// TIA Portal V17 export
// export: Created 2025-03-07T09:18:16.2662316Z, ExportSetting WithDefaults, DisplayName Totally Integrated Automation Portal, DisplayVersion V17 Update 8, DisplayName TIA Portal Openness, DisplayVersion V17 Update 8, DisplayName TIA Portal Version Control Interface, DisplayVersion V17, DisplayName SINAMICS Startdrive Advanced, DisplayVersion V17 SP2, DisplayName SINAMICS Startdrive G110M, G120, G120C, G120D, G120P, G115D, DisplayVersion V17 SP2, DisplayName SINAMICS Startdrive G130, G150, S120, S150, SINAMICS MV, S210, DisplayVersion V17 SP2, DisplayName STEP 7 Professional, DisplayVersion V17 Update 8, DisplayName SINUMERIK ONE STEP 7 Toolbox, DisplayVersion V17 Update 12, DisplayName SINUMERIK 840D sl STEP 7 Toolbox, DisplayVersion V17 Update 12, DisplayName STEP 7 Safety, DisplayVersion V17 Update 6, DisplayName WinCC Advanced, DisplayVersion V17 Update 8
FUNCTION "FC1301_PART_CYCLE_UNIT_03_CLADDING" : Void   // FC1301, LAD
{ S7_Optimized_Access := 'FALSE' }
AUTHOR : ETXETAR
VERSION : 1.0
// stored: AutoNumber false, IsIECCheckEnabled false, SetENOAutomatically false, UDAEnableTagReadback false
   VAR CONSTANT
      FC_NUMBER : DInt := 1301;
   END_VAR
   VAR_TEMP   // added for the SCL form of the ladder/FBD networks
      _w1 : Bool;
      _w2 : Bool;
   END_VAR
BEGIN

REGION Network 1: GENERAL CONDITIONS
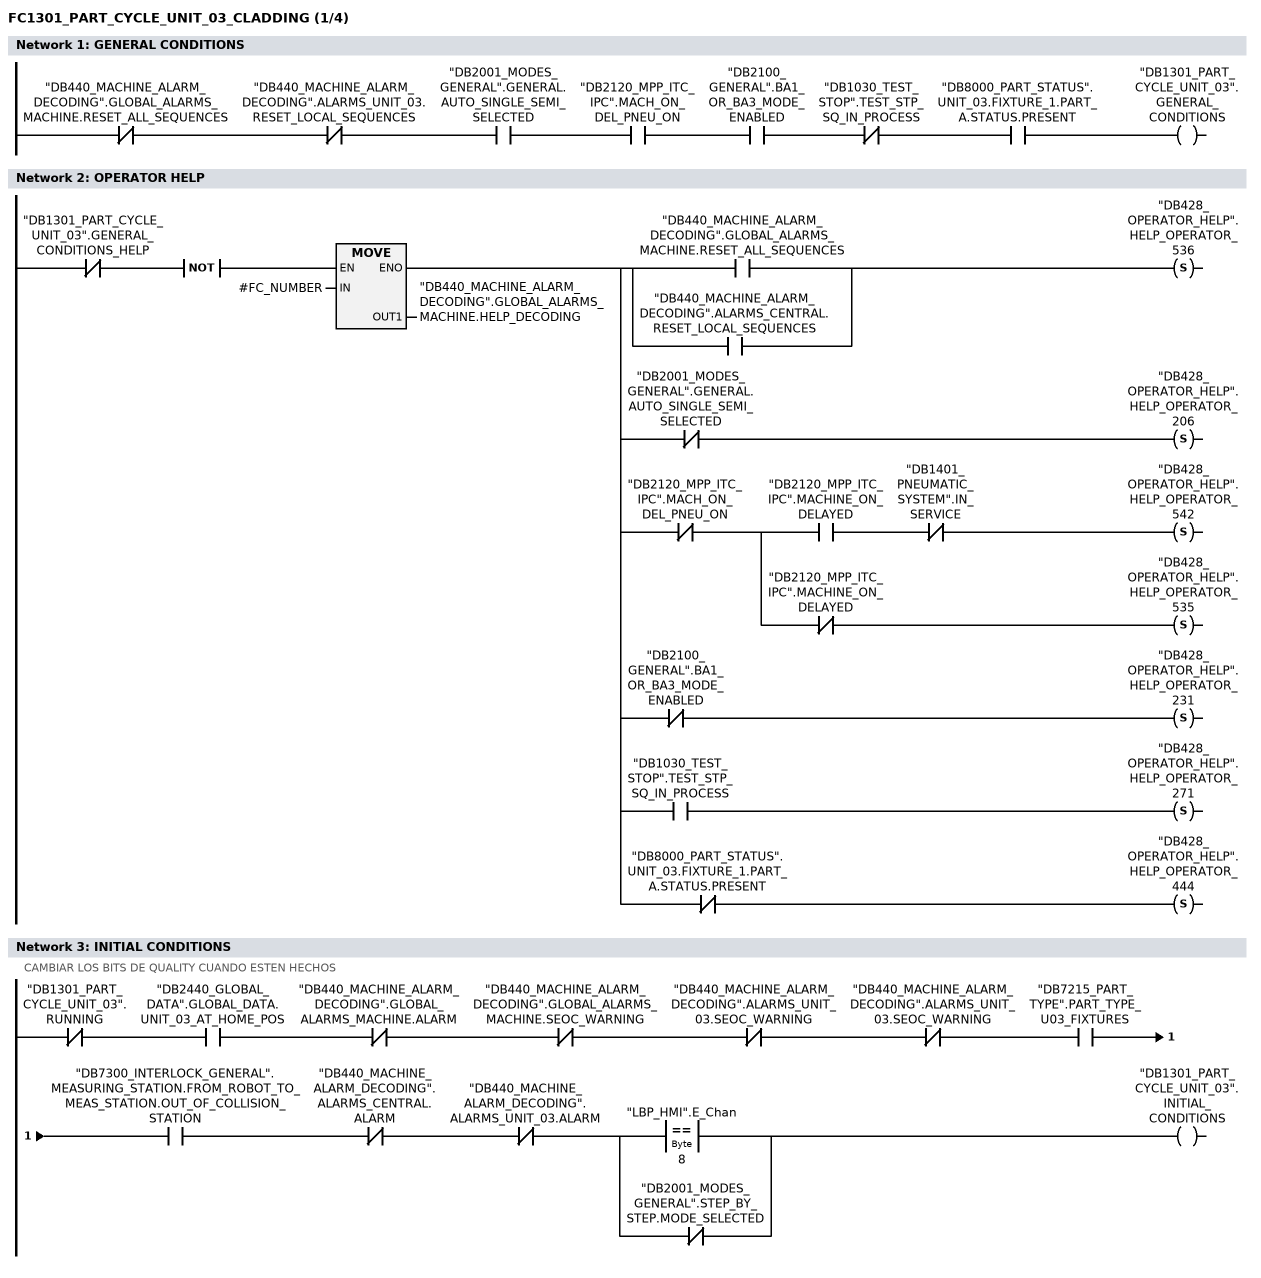
   RUNG wire#powerrail
      I_Contact( "DB440_MACHINE_ALARM_DECODING".GLOBAL_ALARMS_MACHINE.RESET_ALL_SEQUENCES )
      I_Contact( "DB440_MACHINE_ALARM_DECODING".ALARMS_UNIT_03.RESET_LOCAL_SEQUENCES )
      Contact( "DB2001_MODES_GENERAL".GENERAL.AUTO_SINGLE_SEMI_SELECTED )
      Contact( "DB2120_MPP_ITC_IPC".MACH_ON_DEL_PNEU_ON )
      Contact( "DB2100_GENERAL".BA1_OR_BA3_MODE_ENABLED )
      I_Contact( "DB1030_TEST_STOP".TEST_STP_SQ_IN_PROCESS )
      Contact( "DB8000_PART_STATUS".UNIT_03.FIXTURE_1.PART_A.STATUS.PRESENT )
      Coil( "DB1301_PART_CYCLE_UNIT_03".GENERAL_CONDITIONS )
   END_RUNG
   // the same network as SCL:
   "DB1301_PART_CYCLE_UNIT_03".GENERAL_CONDITIONS := NOT "DB440_MACHINE_ALARM_DECODING".GLOBAL_ALARMS_MACHINE.RESET_ALL_SEQUENCES AND NOT "DB440_MACHINE_ALARM_DECODING".ALARMS_UNIT_03.RESET_LOCAL_SEQUENCES AND "DB2001_MODES_GENERAL".GENERAL.AUTO_SINGLE_SEMI_SELECTED AND "DB2120_MPP_ITC_IPC".MACH_ON_DEL_PNEU_ON AND "DB2100_GENERAL".BA1_OR_BA3_MODE_ENABLED AND NOT "DB1030_TEST_STOP".TEST_STP_SQ_IN_PROCESS AND "DB8000_PART_STATUS".UNIT_03.FIXTURE_1.PART_A.STATUS.PRESENT;
END_REGION

REGION Network 2: OPERATOR HELP
   RUNG wire#powerrail
      I_Contact( "DB1301_PART_CYCLE_UNIT_03".GENERAL_CONDITIONS_HELP )
      Not()
      { S7_GenerateENO := "TRUE" } Move(in := #FC_NUMBER, out1 => "DB440_MACHINE_ALARM_DECODING".GLOBAL_ALARMS_MACHINE.HELP_DECODING)
      wire#w1
      Contact( "DB440_MACHINE_ALARM_DECODING".GLOBAL_ALARMS_MACHINE.RESET_ALL_SEQUENCES )
      wire#w2
      S_Coil( "DB428_OPERATOR_HELP".HELP_OPERATOR_536 )
   END_RUNG
   RUNG wire#w1
      Contact( "DB440_MACHINE_ALARM_DECODING".ALARMS_CENTRAL.RESET_LOCAL_SEQUENCES )
   END_RUNG wire#w2
   RUNG wire#w1
      I_Contact( "DB2001_MODES_GENERAL".GENERAL.AUTO_SINGLE_SEMI_SELECTED )
      S_Coil( "DB428_OPERATOR_HELP".HELP_OPERATOR_206 )
   END_RUNG
   RUNG wire#w1
      I_Contact( "DB2120_MPP_ITC_IPC".MACH_ON_DEL_PNEU_ON )
      wire#w3
      Contact( "DB2120_MPP_ITC_IPC".MACHINE_ON_DELAYED )
      I_Contact( "DB1401_PNEUMATIC_SYSTEM".IN_SERVICE )
      S_Coil( "DB428_OPERATOR_HELP".HELP_OPERATOR_542 )
   END_RUNG
   RUNG wire#w3
      I_Contact( "DB2120_MPP_ITC_IPC".MACHINE_ON_DELAYED )
      S_Coil( "DB428_OPERATOR_HELP".HELP_OPERATOR_535 )
   END_RUNG
   RUNG wire#w1
      I_Contact( "DB2100_GENERAL".BA1_OR_BA3_MODE_ENABLED )
      S_Coil( "DB428_OPERATOR_HELP".HELP_OPERATOR_231 )
   END_RUNG
   RUNG wire#w1
      Contact( "DB1030_TEST_STOP".TEST_STP_SQ_IN_PROCESS )
      S_Coil( "DB428_OPERATOR_HELP".HELP_OPERATOR_271 )
   END_RUNG
   RUNG wire#w1
      I_Contact( "DB8000_PART_STATUS".UNIT_03.FIXTURE_1.PART_A.STATUS.PRESENT )
      S_Coil( "DB428_OPERATOR_HELP".HELP_OPERATOR_444 )
   END_RUNG
   // the same network as SCL:
   // ENO of a box is taken as its EN; it also drops when the box reports an error
   #_w1 := NOT (NOT "DB1301_PART_CYCLE_UNIT_03".GENERAL_CONDITIONS_HELP);
   IF #_w1 THEN "DB440_MACHINE_ALARM_DECODING".GLOBAL_ALARMS_MACHINE.HELP_DECODING := #FC_NUMBER; END_IF;
   IF #_w1 AND ("DB440_MACHINE_ALARM_DECODING".GLOBAL_ALARMS_MACHINE.RESET_ALL_SEQUENCES OR "DB440_MACHINE_ALARM_DECODING".ALARMS_CENTRAL.RESET_LOCAL_SEQUENCES) THEN
       "DB428_OPERATOR_HELP".HELP_OPERATOR_536 := TRUE;
   END_IF;
   IF #_w1 AND NOT "DB2001_MODES_GENERAL".GENERAL.AUTO_SINGLE_SEMI_SELECTED THEN
       "DB428_OPERATOR_HELP".HELP_OPERATOR_206 := TRUE;
   END_IF;
   #_w2 := #_w1 AND NOT "DB2120_MPP_ITC_IPC".MACH_ON_DEL_PNEU_ON;
   IF #_w2 AND "DB2120_MPP_ITC_IPC".MACHINE_ON_DELAYED AND NOT "DB1401_PNEUMATIC_SYSTEM".IN_SERVICE THEN
       "DB428_OPERATOR_HELP".HELP_OPERATOR_542 := TRUE;
   END_IF;
   IF #_w2 AND NOT "DB2120_MPP_ITC_IPC".MACHINE_ON_DELAYED THEN
       "DB428_OPERATOR_HELP".HELP_OPERATOR_535 := TRUE;
   END_IF;
   IF #_w1 AND NOT "DB2100_GENERAL".BA1_OR_BA3_MODE_ENABLED THEN
       "DB428_OPERATOR_HELP".HELP_OPERATOR_231 := TRUE;
   END_IF;
   IF #_w1 AND "DB1030_TEST_STOP".TEST_STP_SQ_IN_PROCESS THEN
       "DB428_OPERATOR_HELP".HELP_OPERATOR_271 := TRUE;
   END_IF;
   IF #_w1 AND NOT "DB8000_PART_STATUS".UNIT_03.FIXTURE_1.PART_A.STATUS.PRESENT THEN
       "DB428_OPERATOR_HELP".HELP_OPERATOR_444 := TRUE;
   END_IF;
END_REGION

REGION Network 3: INITIAL CONDITIONS
   // CAMBIAR LOS BITS DE QUALITY CUANDO ESTEN HECHOS
   RUNG wire#powerrail
      I_Contact( "DB1301_PART_CYCLE_UNIT_03".RUNNING )
      Contact( "DB2440_GLOBAL_DATA".GLOBAL_DATA.UNIT_03_AT_HOME_POS )
      I_Contact( "DB440_MACHINE_ALARM_DECODING".GLOBAL_ALARMS_MACHINE.ALARM )
      I_Contact( "DB440_MACHINE_ALARM_DECODING".GLOBAL_ALARMS_MACHINE.SEOC_WARNING )
      I_Contact( "DB440_MACHINE_ALARM_DECODING".ALARMS_UNIT_03.SEOC_WARNING )
      I_Contact( "DB440_MACHINE_ALARM_DECODING".ALARMS_UNIT_03.SEOC_WARNING )
      Contact( "DB7215_PART_TYPE".PART_TYPE_U03_FIXTURES )
      Contact( "DB7300_INTERLOCK_GENERAL".MEASURING_STATION.FROM_ROBOT_TO_MEAS_STATION.OUT_OF_COLLISION_STATION )
      I_Contact( "DB440_MACHINE_ALARM_DECODING".ALARMS_CENTRAL.ALARM )
      I_Contact( "DB440_MACHINE_ALARM_DECODING".ALARMS_UNIT_03.ALARM )
      wire#w1
      { S7_Templates := "SrcType := Byte" } EQ_Contact(in1 := "LBP_HMI".E_Chan, in2 := 8)
      wire#w2
      Coil( "DB1301_PART_CYCLE_UNIT_03".INITIAL_CONDITIONS )
   END_RUNG
   RUNG wire#w1
      I_Contact( "DB2001_MODES_GENERAL".STEP_BY_STEP.MODE_SELECTED )
   END_RUNG wire#w2
   // the same network as SCL:
   "DB1301_PART_CYCLE_UNIT_03".INITIAL_CONDITIONS := NOT "DB1301_PART_CYCLE_UNIT_03".RUNNING AND "DB2440_GLOBAL_DATA".GLOBAL_DATA.UNIT_03_AT_HOME_POS AND NOT "DB440_MACHINE_ALARM_DECODING".GLOBAL_ALARMS_MACHINE.ALARM AND NOT "DB440_MACHINE_ALARM_DECODING".GLOBAL_ALARMS_MACHINE.SEOC_WARNING AND NOT "DB440_MACHINE_ALARM_DECODING".ALARMS_UNIT_03.SEOC_WARNING AND NOT "DB440_MACHINE_ALARM_DECODING".ALARMS_UNIT_03.SEOC_WARNING AND "DB7215_PART_TYPE".PART_TYPE_U03_FIXTURES AND "DB7300_INTERLOCK_GENERAL".MEASURING_STATION.FROM_ROBOT_TO_MEAS_STATION.OUT_OF_COLLISION_STATION AND NOT "DB440_MACHINE_ALARM_DECODING".ALARMS_CENTRAL.ALARM AND NOT "DB440_MACHINE_ALARM_DECODING".ALARMS_UNIT_03.ALARM AND (("LBP_HMI".E_Chan = 8) OR NOT "DB2001_MODES_GENERAL".STEP_BY_STEP.MODE_SELECTED);
END_REGION

REGION Network 4: OPERATOR HELP
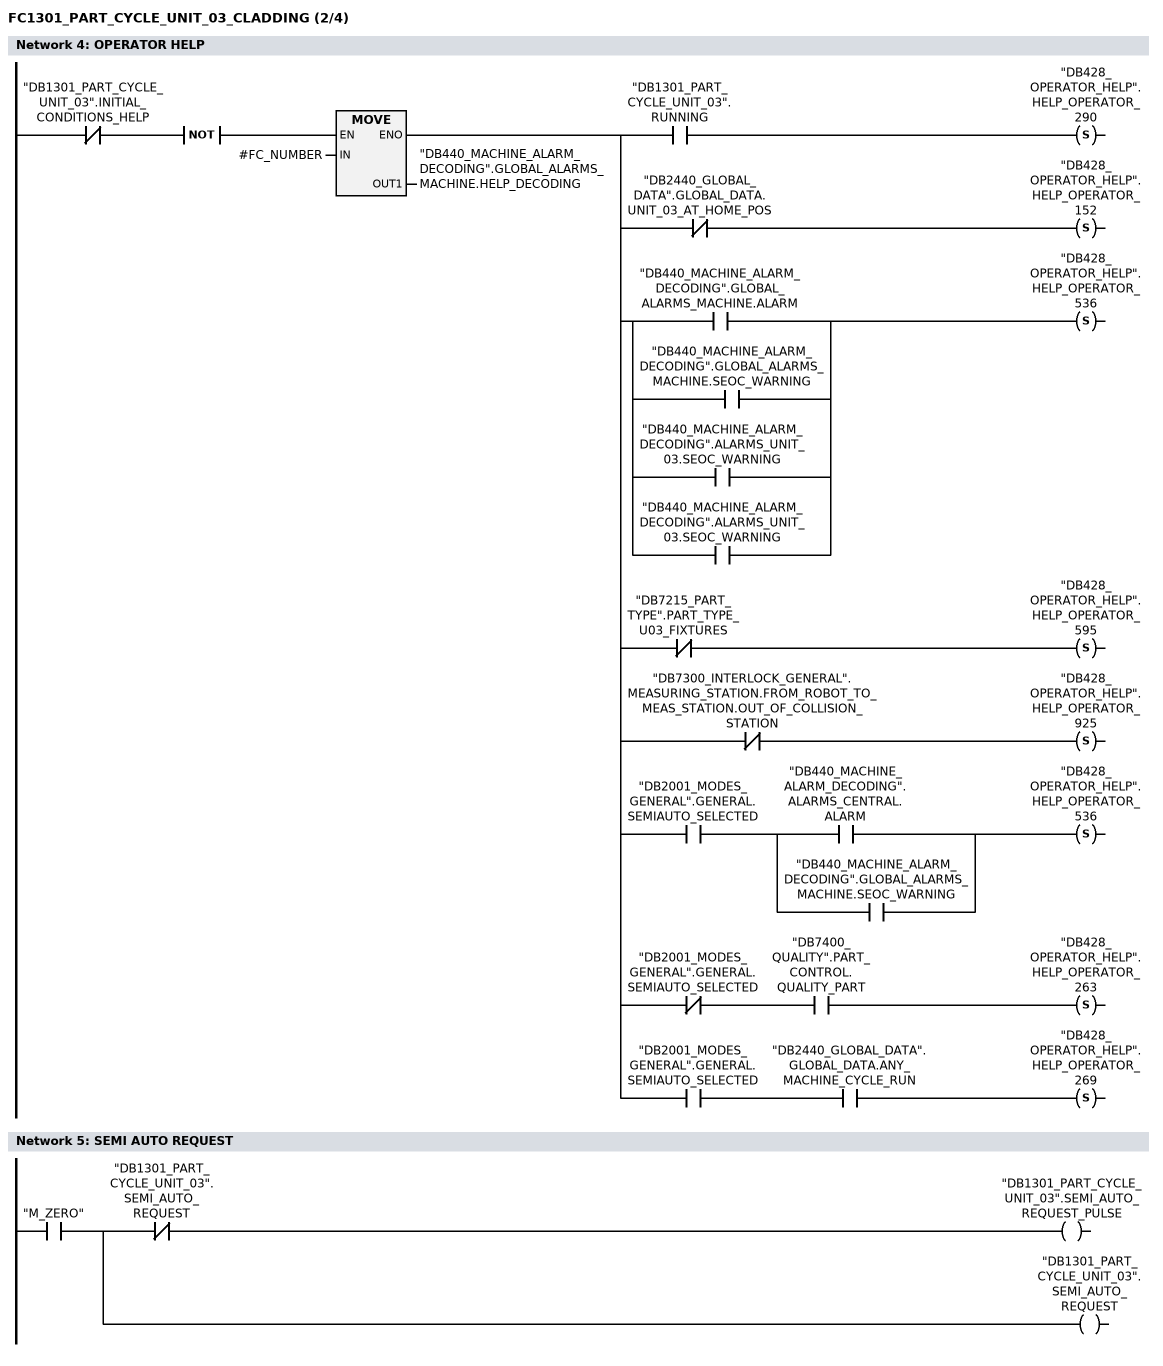
   RUNG wire#powerrail
      I_Contact( "DB1301_PART_CYCLE_UNIT_03".INITIAL_CONDITIONS_HELP )
      Not()
      { S7_GenerateENO := "TRUE" } Move(in := #FC_NUMBER, out1 => "DB440_MACHINE_ALARM_DECODING".GLOBAL_ALARMS_MACHINE.HELP_DECODING)
      wire#w1
      Contact( "DB1301_PART_CYCLE_UNIT_03".RUNNING )
      S_Coil( "DB428_OPERATOR_HELP".HELP_OPERATOR_290 )
   END_RUNG
   RUNG wire#w1
      I_Contact( "DB2440_GLOBAL_DATA".GLOBAL_DATA.UNIT_03_AT_HOME_POS )
      S_Coil( "DB428_OPERATOR_HELP".HELP_OPERATOR_152 )
   END_RUNG
   RUNG wire#w1
      Contact( "DB440_MACHINE_ALARM_DECODING".GLOBAL_ALARMS_MACHINE.ALARM )
      wire#w2
      S_Coil( "DB428_OPERATOR_HELP".HELP_OPERATOR_536 )
   END_RUNG
   RUNG wire#w1
      Contact( "DB440_MACHINE_ALARM_DECODING".GLOBAL_ALARMS_MACHINE.SEOC_WARNING )
   END_RUNG wire#w2
   RUNG wire#w1
      Contact( "DB440_MACHINE_ALARM_DECODING".ALARMS_UNIT_03.SEOC_WARNING )
   END_RUNG wire#w2
   RUNG wire#w1
      Contact( "DB440_MACHINE_ALARM_DECODING".ALARMS_UNIT_03.SEOC_WARNING )
   END_RUNG wire#w2
   RUNG wire#w1
      I_Contact( "DB7215_PART_TYPE".PART_TYPE_U03_FIXTURES )
      S_Coil( "DB428_OPERATOR_HELP".HELP_OPERATOR_595 )
   END_RUNG
   RUNG wire#w1
      I_Contact( "DB7300_INTERLOCK_GENERAL".MEASURING_STATION.FROM_ROBOT_TO_MEAS_STATION.OUT_OF_COLLISION_STATION )
      S_Coil( "DB428_OPERATOR_HELP".HELP_OPERATOR_925 )
   END_RUNG
   RUNG wire#w1
      Contact( "DB2001_MODES_GENERAL".GENERAL.SEMIAUTO_SELECTED )
      wire#w3
      Contact( "DB440_MACHINE_ALARM_DECODING".ALARMS_CENTRAL.ALARM )
      wire#w4
      S_Coil( "DB428_OPERATOR_HELP".HELP_OPERATOR_536 )
   END_RUNG
   RUNG wire#w3
      Contact( "DB440_MACHINE_ALARM_DECODING".GLOBAL_ALARMS_MACHINE.SEOC_WARNING )
   END_RUNG wire#w4
   RUNG wire#w1
      I_Contact( "DB2001_MODES_GENERAL".GENERAL.SEMIAUTO_SELECTED )
      Contact( "DB7400_QUALITY".PART_CONTROL.QUALITY_PART )
      S_Coil( "DB428_OPERATOR_HELP".HELP_OPERATOR_263 )
   END_RUNG
   RUNG wire#w1
      Contact( "DB2001_MODES_GENERAL".GENERAL.SEMIAUTO_SELECTED )
      Contact( "DB2440_GLOBAL_DATA".GLOBAL_DATA.ANY_MACHINE_CYCLE_RUN )
      S_Coil( "DB428_OPERATOR_HELP".HELP_OPERATOR_269 )
   END_RUNG
   // the same network as SCL:
   // ENO of a box is taken as its EN; it also drops when the box reports an error
   #_w1 := NOT (NOT "DB1301_PART_CYCLE_UNIT_03".INITIAL_CONDITIONS_HELP);
   IF #_w1 THEN "DB440_MACHINE_ALARM_DECODING".GLOBAL_ALARMS_MACHINE.HELP_DECODING := #FC_NUMBER; END_IF;
   IF #_w1 AND "DB1301_PART_CYCLE_UNIT_03".RUNNING THEN
       "DB428_OPERATOR_HELP".HELP_OPERATOR_290 := TRUE;
   END_IF;
   IF #_w1 AND NOT "DB2440_GLOBAL_DATA".GLOBAL_DATA.UNIT_03_AT_HOME_POS THEN
       "DB428_OPERATOR_HELP".HELP_OPERATOR_152 := TRUE;
   END_IF;
   IF #_w1 AND ("DB440_MACHINE_ALARM_DECODING".GLOBAL_ALARMS_MACHINE.ALARM OR "DB440_MACHINE_ALARM_DECODING".GLOBAL_ALARMS_MACHINE.SEOC_WARNING OR "DB440_MACHINE_ALARM_DECODING".ALARMS_UNIT_03.SEOC_WARNING OR "DB440_MACHINE_ALARM_DECODING".ALARMS_UNIT_03.SEOC_WARNING) THEN
       "DB428_OPERATOR_HELP".HELP_OPERATOR_536 := TRUE;
   END_IF;
   IF #_w1 AND NOT "DB7215_PART_TYPE".PART_TYPE_U03_FIXTURES THEN
       "DB428_OPERATOR_HELP".HELP_OPERATOR_595 := TRUE;
   END_IF;
   IF #_w1 AND NOT "DB7300_INTERLOCK_GENERAL".MEASURING_STATION.FROM_ROBOT_TO_MEAS_STATION.OUT_OF_COLLISION_STATION THEN
       "DB428_OPERATOR_HELP".HELP_OPERATOR_925 := TRUE;
   END_IF;
   IF #_w1 AND "DB2001_MODES_GENERAL".GENERAL.SEMIAUTO_SELECTED AND ("DB440_MACHINE_ALARM_DECODING".ALARMS_CENTRAL.ALARM OR "DB440_MACHINE_ALARM_DECODING".GLOBAL_ALARMS_MACHINE.SEOC_WARNING) THEN
       "DB428_OPERATOR_HELP".HELP_OPERATOR_536 := TRUE;
   END_IF;
   IF #_w1 AND NOT "DB2001_MODES_GENERAL".GENERAL.SEMIAUTO_SELECTED AND "DB7400_QUALITY".PART_CONTROL.QUALITY_PART THEN
       "DB428_OPERATOR_HELP".HELP_OPERATOR_263 := TRUE;
   END_IF;
   IF #_w1 AND "DB2001_MODES_GENERAL".GENERAL.SEMIAUTO_SELECTED AND "DB2440_GLOBAL_DATA".GLOBAL_DATA.ANY_MACHINE_CYCLE_RUN THEN
       "DB428_OPERATOR_HELP".HELP_OPERATOR_269 := TRUE;
   END_IF;
END_REGION

REGION Network 5: SEMI AUTO REQUEST
   RUNG wire#powerrail
      Contact( "M_ZERO" )
      wire#w1
      I_Contact( "DB1301_PART_CYCLE_UNIT_03".SEMI_AUTO_REQUEST )
      Coil( "DB1301_PART_CYCLE_UNIT_03".SEMI_AUTO_REQUEST_PULSE )
   END_RUNG
   RUNG wire#w1
      Coil( "DB1301_PART_CYCLE_UNIT_03".SEMI_AUTO_REQUEST )
   END_RUNG
   // the same network as SCL:
   "DB1301_PART_CYCLE_UNIT_03".SEMI_AUTO_REQUEST_PULSE := "M_ZERO" AND NOT "DB1301_PART_CYCLE_UNIT_03".SEMI_AUTO_REQUEST;
   "DB1301_PART_CYCLE_UNIT_03".SEMI_AUTO_REQUEST := "M_ZERO";
END_REGION

REGION Network 6: OPERATOR HELP
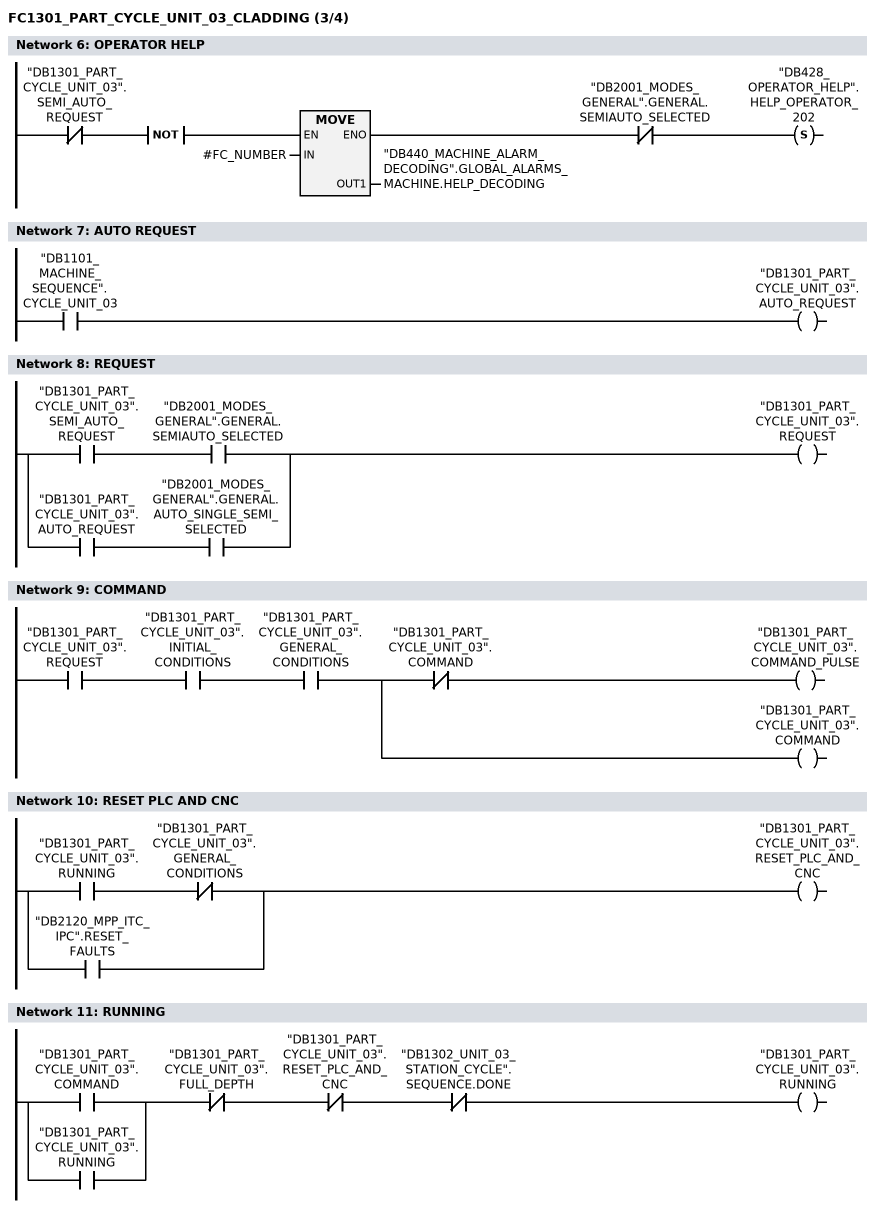
   RUNG wire#powerrail
      I_Contact( "DB1301_PART_CYCLE_UNIT_03".SEMI_AUTO_REQUEST )
      Not()
      { S7_GenerateENO := "TRUE" } Move(in := #FC_NUMBER, out1 => "DB440_MACHINE_ALARM_DECODING".GLOBAL_ALARMS_MACHINE.HELP_DECODING)
      I_Contact( "DB2001_MODES_GENERAL".GENERAL.SEMIAUTO_SELECTED )
      S_Coil( "DB428_OPERATOR_HELP".HELP_OPERATOR_202 )
   END_RUNG
   // the same network as SCL:
   // ENO of a box is taken as its EN; it also drops when the box reports an error
   #_w1 := NOT (NOT "DB1301_PART_CYCLE_UNIT_03".SEMI_AUTO_REQUEST);
   IF #_w1 THEN "DB440_MACHINE_ALARM_DECODING".GLOBAL_ALARMS_MACHINE.HELP_DECODING := #FC_NUMBER; END_IF;
   IF #_w1 AND NOT "DB2001_MODES_GENERAL".GENERAL.SEMIAUTO_SELECTED THEN
       "DB428_OPERATOR_HELP".HELP_OPERATOR_202 := TRUE;
   END_IF;
END_REGION

REGION Network 7: AUTO REQUEST
   RUNG wire#powerrail
      Contact( "DB1101_MACHINE_SEQUENCE".CYCLE_UNIT_03 )
      Coil( "DB1301_PART_CYCLE_UNIT_03".AUTO_REQUEST )
   END_RUNG
   // the same network as SCL:
   "DB1301_PART_CYCLE_UNIT_03".AUTO_REQUEST := "DB1101_MACHINE_SEQUENCE".CYCLE_UNIT_03;
END_REGION

REGION Network 8: REQUEST
   RUNG wire#powerrail
      Contact( "DB1301_PART_CYCLE_UNIT_03".SEMI_AUTO_REQUEST )
      Contact( "DB2001_MODES_GENERAL".GENERAL.SEMIAUTO_SELECTED )
      wire#w1
      Coil( "DB1301_PART_CYCLE_UNIT_03".REQUEST )
   END_RUNG
   RUNG wire#powerrail
      Contact( "DB1301_PART_CYCLE_UNIT_03".AUTO_REQUEST )
      Contact( "DB2001_MODES_GENERAL".GENERAL.AUTO_SINGLE_SEMI_SELECTED )
   END_RUNG wire#w1
   // the same network as SCL:
   "DB1301_PART_CYCLE_UNIT_03".REQUEST := ("DB1301_PART_CYCLE_UNIT_03".SEMI_AUTO_REQUEST AND "DB2001_MODES_GENERAL".GENERAL.SEMIAUTO_SELECTED) OR ("DB1301_PART_CYCLE_UNIT_03".AUTO_REQUEST AND "DB2001_MODES_GENERAL".GENERAL.AUTO_SINGLE_SEMI_SELECTED);
END_REGION

REGION Network 9: COMMAND
   RUNG wire#powerrail
      Contact( "DB1301_PART_CYCLE_UNIT_03".REQUEST )
      Contact( "DB1301_PART_CYCLE_UNIT_03".INITIAL_CONDITIONS )
      Contact( "DB1301_PART_CYCLE_UNIT_03".GENERAL_CONDITIONS )
      wire#w1
      I_Contact( "DB1301_PART_CYCLE_UNIT_03".COMMAND )
      Coil( "DB1301_PART_CYCLE_UNIT_03".COMMAND_PULSE )
   END_RUNG
   RUNG wire#w1
      Coil( "DB1301_PART_CYCLE_UNIT_03".COMMAND )
   END_RUNG
   // the same network as SCL:
   #_w1 := "DB1301_PART_CYCLE_UNIT_03".REQUEST AND "DB1301_PART_CYCLE_UNIT_03".INITIAL_CONDITIONS AND "DB1301_PART_CYCLE_UNIT_03".GENERAL_CONDITIONS;
   "DB1301_PART_CYCLE_UNIT_03".COMMAND_PULSE := #_w1 AND NOT "DB1301_PART_CYCLE_UNIT_03".COMMAND;
   "DB1301_PART_CYCLE_UNIT_03".COMMAND := #_w1;
END_REGION

REGION Network 10: RESET PLC AND CNC
   RUNG wire#powerrail
      Contact( "DB1301_PART_CYCLE_UNIT_03".RUNNING )
      I_Contact( "DB1301_PART_CYCLE_UNIT_03".GENERAL_CONDITIONS )
      wire#w1
      Coil( "DB1301_PART_CYCLE_UNIT_03".RESET_PLC_AND_CNC )
   END_RUNG
   RUNG wire#powerrail
      Contact( "DB2120_MPP_ITC_IPC".RESET_FAULTS )
   END_RUNG wire#w1
   // the same network as SCL:
   "DB1301_PART_CYCLE_UNIT_03".RESET_PLC_AND_CNC := ("DB1301_PART_CYCLE_UNIT_03".RUNNING AND NOT "DB1301_PART_CYCLE_UNIT_03".GENERAL_CONDITIONS) OR "DB2120_MPP_ITC_IPC".RESET_FAULTS;
END_REGION

REGION Network 11: RUNNING
   RUNG wire#powerrail
      Contact( "DB1301_PART_CYCLE_UNIT_03".COMMAND )
      wire#w1
      I_Contact( "DB1301_PART_CYCLE_UNIT_03".FULL_DEPTH )
      I_Contact( "DB1301_PART_CYCLE_UNIT_03".RESET_PLC_AND_CNC )
      I_Contact( "DB1302_UNIT_03_STATION_CYCLE".SEQUENCE.DONE )
      Coil( "DB1301_PART_CYCLE_UNIT_03".RUNNING )
   END_RUNG
   RUNG wire#powerrail
      Contact( "DB1301_PART_CYCLE_UNIT_03".RUNNING )
   END_RUNG wire#w1
   // the same network as SCL:
   "DB1301_PART_CYCLE_UNIT_03".RUNNING := ("DB1301_PART_CYCLE_UNIT_03".COMMAND OR "DB1301_PART_CYCLE_UNIT_03".RUNNING) AND NOT "DB1301_PART_CYCLE_UNIT_03".FULL_DEPTH AND NOT "DB1301_PART_CYCLE_UNIT_03".RESET_PLC_AND_CNC AND NOT "DB1302_UNIT_03_STATION_CYCLE".SEQUENCE.DONE;
END_REGION

REGION Network 12: CYCLE MEASURE UNIT STATION
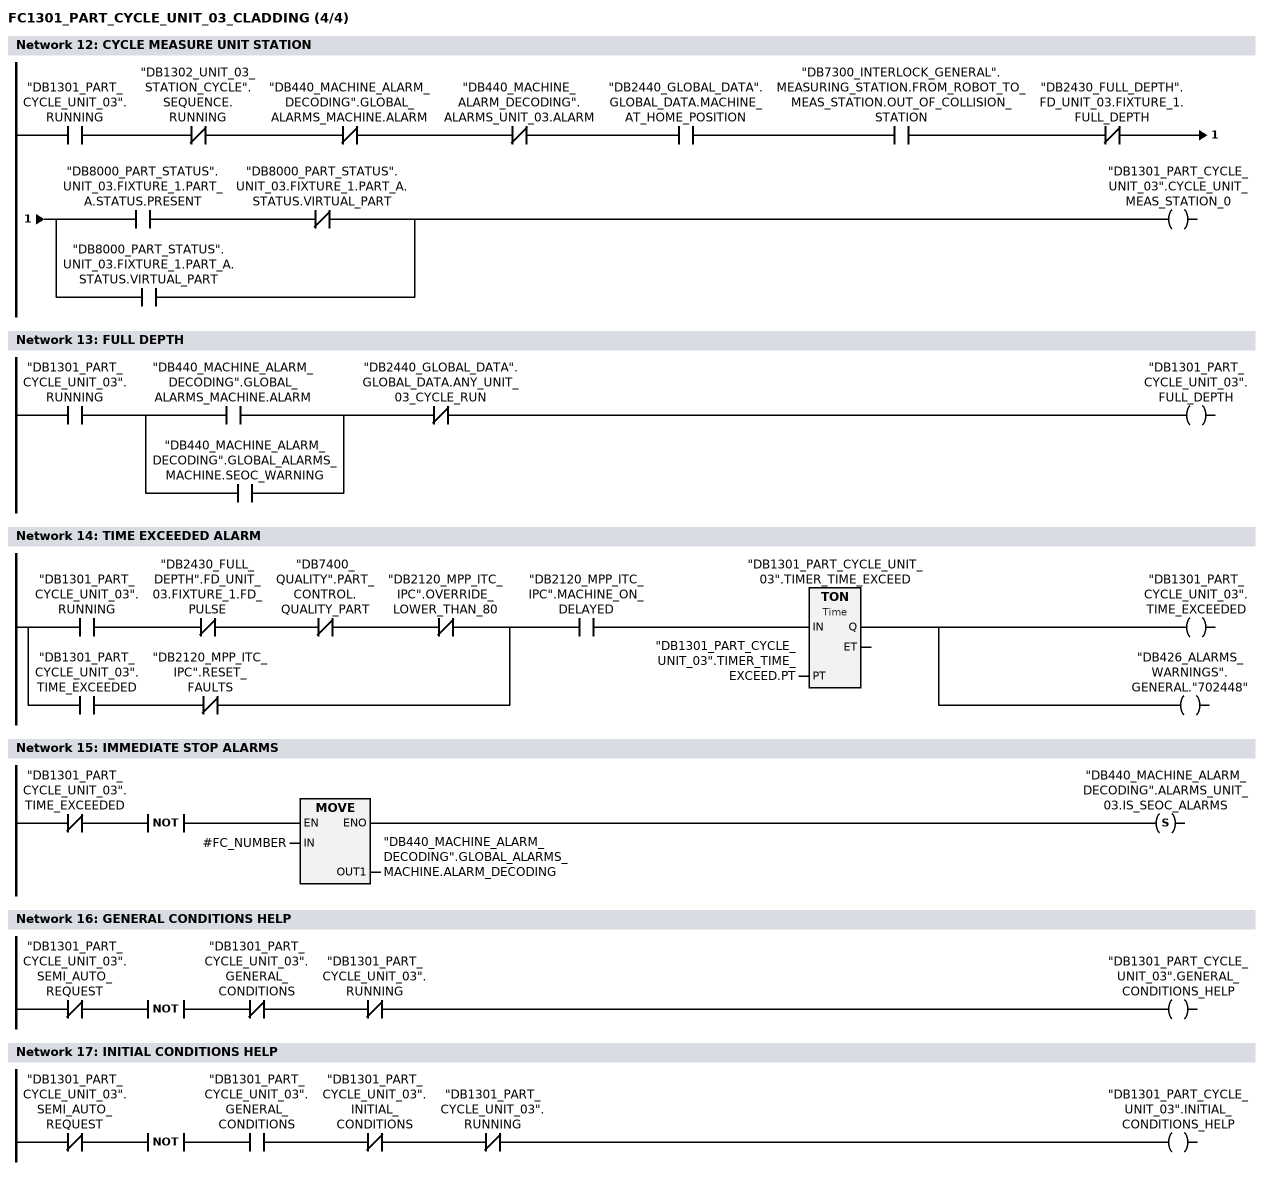
   RUNG wire#powerrail
      Contact( "DB1301_PART_CYCLE_UNIT_03".RUNNING )
      I_Contact( "DB1302_UNIT_03_STATION_CYCLE".SEQUENCE.RUNNING )
      I_Contact( "DB440_MACHINE_ALARM_DECODING".GLOBAL_ALARMS_MACHINE.ALARM )
      I_Contact( "DB440_MACHINE_ALARM_DECODING".ALARMS_UNIT_03.ALARM )
      Contact( "DB2440_GLOBAL_DATA".GLOBAL_DATA.MACHINE_AT_HOME_POSITION )
      Contact( "DB7300_INTERLOCK_GENERAL".MEASURING_STATION.FROM_ROBOT_TO_MEAS_STATION.OUT_OF_COLLISION_STATION )
      I_Contact( "DB2430_FULL_DEPTH".FD_UNIT_03.FIXTURE_1.FULL_DEPTH )
      wire#w1
      Contact( "DB8000_PART_STATUS".UNIT_03.FIXTURE_1.PART_A.STATUS.PRESENT )
      I_Contact( "DB8000_PART_STATUS".UNIT_03.FIXTURE_1.PART_A.STATUS.VIRTUAL_PART )
      wire#w2
      Coil( "DB1301_PART_CYCLE_UNIT_03".CYCLE_UNIT_MEAS_STATION_0 )
   END_RUNG
   RUNG wire#w1
      Contact( "DB8000_PART_STATUS".UNIT_03.FIXTURE_1.PART_A.STATUS.VIRTUAL_PART )
   END_RUNG wire#w2
   // the same network as SCL:
   "DB1301_PART_CYCLE_UNIT_03".CYCLE_UNIT_MEAS_STATION_0 := "DB1301_PART_CYCLE_UNIT_03".RUNNING AND NOT "DB1302_UNIT_03_STATION_CYCLE".SEQUENCE.RUNNING AND NOT "DB440_MACHINE_ALARM_DECODING".GLOBAL_ALARMS_MACHINE.ALARM AND NOT "DB440_MACHINE_ALARM_DECODING".ALARMS_UNIT_03.ALARM AND "DB2440_GLOBAL_DATA".GLOBAL_DATA.MACHINE_AT_HOME_POSITION AND "DB7300_INTERLOCK_GENERAL".MEASURING_STATION.FROM_ROBOT_TO_MEAS_STATION.OUT_OF_COLLISION_STATION AND NOT "DB2430_FULL_DEPTH".FD_UNIT_03.FIXTURE_1.FULL_DEPTH AND (("DB8000_PART_STATUS".UNIT_03.FIXTURE_1.PART_A.STATUS.PRESENT AND NOT "DB8000_PART_STATUS".UNIT_03.FIXTURE_1.PART_A.STATUS.VIRTUAL_PART) OR "DB8000_PART_STATUS".UNIT_03.FIXTURE_1.PART_A.STATUS.VIRTUAL_PART);
END_REGION

REGION Network 13: FULL DEPTH
   RUNG wire#powerrail
      Contact( "DB1301_PART_CYCLE_UNIT_03".RUNNING )
      wire#w1
      Contact( "DB440_MACHINE_ALARM_DECODING".GLOBAL_ALARMS_MACHINE.ALARM )
      wire#w2
      I_Contact( "DB2440_GLOBAL_DATA".GLOBAL_DATA.ANY_UNIT_03_CYCLE_RUN )
      Coil( "DB1301_PART_CYCLE_UNIT_03".FULL_DEPTH )
   END_RUNG
   RUNG wire#w1
      Contact( "DB440_MACHINE_ALARM_DECODING".GLOBAL_ALARMS_MACHINE.SEOC_WARNING )
   END_RUNG wire#w2
   // the same network as SCL:
   "DB1301_PART_CYCLE_UNIT_03".FULL_DEPTH := "DB1301_PART_CYCLE_UNIT_03".RUNNING AND ("DB440_MACHINE_ALARM_DECODING".GLOBAL_ALARMS_MACHINE.ALARM OR "DB440_MACHINE_ALARM_DECODING".GLOBAL_ALARMS_MACHINE.SEOC_WARNING) AND NOT "DB2440_GLOBAL_DATA".GLOBAL_DATA.ANY_UNIT_03_CYCLE_RUN;
END_REGION

REGION Network 14: TIME EXCEEDED ALARM
   RUNG wire#powerrail
      Contact( "DB1301_PART_CYCLE_UNIT_03".RUNNING )
      I_Contact( "DB2430_FULL_DEPTH".FD_UNIT_03.FIXTURE_1.FD_PULSE )
      I_Contact( "DB7400_QUALITY".PART_CONTROL.QUALITY_PART )
      I_Contact( "DB2120_MPP_ITC_IPC".OVERRIDE_LOWER_THAN_80 )
      wire#w1
      Contact( "DB2120_MPP_ITC_IPC".MACHINE_ON_DELAYED )
      { S7_Templates := "time_type := Time" } "DB1301_PART_CYCLE_UNIT_03".TIMER_TIME_EXCEED.TON(pt := "DB1301_PART_CYCLE_UNIT_03".TIMER_TIME_EXCEED.PT, et =>)
      wire#w2
      Coil( "DB1301_PART_CYCLE_UNIT_03".TIME_EXCEEDED )
   END_RUNG
   RUNG wire#powerrail
      Contact( "DB1301_PART_CYCLE_UNIT_03".TIME_EXCEEDED )
      I_Contact( "DB2120_MPP_ITC_IPC".RESET_FAULTS )
   END_RUNG wire#w1
   RUNG wire#w2
      Coil( "DB426_ALARMS_WARNINGS".GENERAL."702448" )
   END_RUNG
   // the same network as SCL:
   "DB1301_PART_CYCLE_UNIT_03".TIMER_TIME_EXCEED.TON(IN := (("DB1301_PART_CYCLE_UNIT_03".RUNNING AND NOT "DB2430_FULL_DEPTH".FD_UNIT_03.FIXTURE_1.FD_PULSE AND NOT "DB7400_QUALITY".PART_CONTROL.QUALITY_PART AND NOT "DB2120_MPP_ITC_IPC".OVERRIDE_LOWER_THAN_80) OR ("DB1301_PART_CYCLE_UNIT_03".TIME_EXCEEDED AND NOT "DB2120_MPP_ITC_IPC".RESET_FAULTS)) AND "DB2120_MPP_ITC_IPC".MACHINE_ON_DELAYED,
                           PT := "DB1301_PART_CYCLE_UNIT_03".TIMER_TIME_EXCEED.PT);
   "DB1301_PART_CYCLE_UNIT_03".TIME_EXCEEDED := "DB1301_PART_CYCLE_UNIT_03".TIMER_TIME_EXCEED.Q;
   "DB426_ALARMS_WARNINGS".GENERAL."702448" := "DB1301_PART_CYCLE_UNIT_03".TIMER_TIME_EXCEED.Q;
END_REGION

REGION Network 15: IMMEDIATE STOP ALARMS
   RUNG wire#powerrail
      I_Contact( "DB1301_PART_CYCLE_UNIT_03".TIME_EXCEEDED )
      Not()
      { S7_GenerateENO := "TRUE" } Move(in := #FC_NUMBER, out1 => "DB440_MACHINE_ALARM_DECODING".GLOBAL_ALARMS_MACHINE.ALARM_DECODING)
      S_Coil( "DB440_MACHINE_ALARM_DECODING".ALARMS_UNIT_03.IS_SEOC_ALARMS )
   END_RUNG
   // the same network as SCL:
   // ENO of a box is taken as its EN; it also drops when the box reports an error
   IF NOT (NOT "DB1301_PART_CYCLE_UNIT_03".TIME_EXCEEDED) THEN
       "DB440_MACHINE_ALARM_DECODING".GLOBAL_ALARMS_MACHINE.ALARM_DECODING := #FC_NUMBER;
       "DB440_MACHINE_ALARM_DECODING".ALARMS_UNIT_03.IS_SEOC_ALARMS := TRUE;
   END_IF;
END_REGION

REGION Network 16: GENERAL CONDITIONS HELP
   RUNG wire#powerrail
      I_Contact( "DB1301_PART_CYCLE_UNIT_03".SEMI_AUTO_REQUEST )
      Not()
      I_Contact( "DB1301_PART_CYCLE_UNIT_03".GENERAL_CONDITIONS )
      I_Contact( "DB1301_PART_CYCLE_UNIT_03".RUNNING )
      Coil( "DB1301_PART_CYCLE_UNIT_03".GENERAL_CONDITIONS_HELP )
   END_RUNG
   // the same network as SCL:
   "DB1301_PART_CYCLE_UNIT_03".GENERAL_CONDITIONS_HELP := NOT (NOT "DB1301_PART_CYCLE_UNIT_03".SEMI_AUTO_REQUEST) AND NOT "DB1301_PART_CYCLE_UNIT_03".GENERAL_CONDITIONS AND NOT "DB1301_PART_CYCLE_UNIT_03".RUNNING;
END_REGION

REGION Network 17: INITIAL CONDITIONS HELP
   RUNG wire#powerrail
      I_Contact( "DB1301_PART_CYCLE_UNIT_03".SEMI_AUTO_REQUEST )
      Not()
      Contact( "DB1301_PART_CYCLE_UNIT_03".GENERAL_CONDITIONS )
      I_Contact( "DB1301_PART_CYCLE_UNIT_03".INITIAL_CONDITIONS )
      I_Contact( "DB1301_PART_CYCLE_UNIT_03".RUNNING )
      Coil( "DB1301_PART_CYCLE_UNIT_03".INITIAL_CONDITIONS_HELP )
   END_RUNG
   // the same network as SCL:
   "DB1301_PART_CYCLE_UNIT_03".INITIAL_CONDITIONS_HELP := NOT (NOT "DB1301_PART_CYCLE_UNIT_03".SEMI_AUTO_REQUEST) AND "DB1301_PART_CYCLE_UNIT_03".GENERAL_CONDITIONS AND NOT "DB1301_PART_CYCLE_UNIT_03".INITIAL_CONDITIONS AND NOT "DB1301_PART_CYCLE_UNIT_03".RUNNING;
END_REGION
END_FUNCTION
